TYPE U_Word :
UNION
	nWord	: WORD;
	aBytes	: ARRAY[0..1] OF BYTE;
END_UNION
END_TYPE

(* stored: Version 1.1.0.1, ProductVersion 3.1.4024.12
   DUT U_Word: Id {414b420f-2925-446c-8524-152e5372000d} *)
